TEXTLIST EL1904_M_4
  1 = 'interlock_out_right_door' | chinese: 'OUT_右侧门' | Chinese: 'OUT_右侧门'
  2 = 'interlock_out_right_door' | chinese: 'OUT_右侧门' | Chinese: 'OUT_右侧门'
  3 = 'Reset' | chinese: '复位' | Chinese: '复位'
  4 = ''
   = ''
END_TEXTLIST

(* stored: Version 1.1.0.1, ProductVersion 3.1.4024.11
   TextList EL1904_M_4: Id {f5b3bebd-e20e-43f9-9c56-22be41532194} *)
